// TIA Portal V17 export
// export: Created 2025-03-10T12:18:29.0033424Z, ExportSetting WithDefaults, DisplayName Totally Integrated Automation Portal, DisplayVersion V17 Update 8, DisplayName TIA Portal Openness, DisplayVersion V17 Update 8, DisplayName TIA Portal Version Control Interface, DisplayVersion V17, DisplayName SINAMICS Startdrive Advanced, DisplayVersion V17 SP2, DisplayName SINAMICS Startdrive G110M, G120, G120C, G120D, G120P, G115D, DisplayVersion V17 SP2, DisplayName SINAMICS Startdrive G130, G150, S120, S150, SINAMICS MV, S210, DisplayVersion V17 SP2, DisplayName STEP 7 Professional, DisplayVersion V17 Update 8, DisplayName SINUMERIK ONE STEP 7 Toolbox, DisplayVersion V17 Update 12, DisplayName SINUMERIK 840D sl STEP 7 Toolbox, DisplayVersion V17 Update 12, DisplayName STEP 7 Safety, DisplayVersion V17 Update 6, DisplayName WinCC Advanced, DisplayVersion V17 Update 8
DATA_BLOCK "DB2031_CYCLES_GENERAL"   // DB2031
{ S7_Optimized_Access := 'FALSE'; DB_Accessible_From_OPC_UA := 'FALSE' }
AUTHOR : ETXETAR
VERSION : 1.0
// stored: AutoNumber false, DBAccessibleFromOPCUA false, DBAccessibleFromWebserver true, IsOnlyStoredInLoadMemory false, IsWriteProtectedInAS false
   VAR RETAIN
      DRY_CYCLE { S7_SetPoint := 'True'} : "CYCLES";
      MANUAL_LOAD_CYCLE { S7_SetPoint := 'True'} : "CYCLES";
   END_VAR
BEGIN
   // DRY_CYCLE.CYCLE_SELECTED : DRY CYCLE SELECTED
   // DRY_CYCLE.CYCLE_COMPLETED : DRY CYCLE COMPLETED
   // MANUAL_LOAD_CYCLE.CYCLE_SELECTED : MANUAL LOAD CYCLE SELECTED
   // MANUAL_LOAD_CYCLE.CYCLE_COMPLETED : MANUAL LOAD CYCLE COMPLETED
END_DATA_BLOCK
